// TIA Portal V17 export
// export: Created 2022-01-31T14:44:44.9197147Z, ExportSetting WithDefaults, DisplayName Totally Integrated Automation Portal, DisplayVersion V17, DisplayName TIA Portal Openness, DisplayVersion V17, DisplayName TIA Portal Version Control Interface, DisplayVersion V17, DisplayName STEP 7 Professional, DisplayVersion V17, DisplayName STEP 7 Safety, DisplayVersion V17, DisplayName WinCC Professional, DisplayVersion V17
DATA_BLOCK "FB_Condensador_DB"   // DB8
VERSION : 0.1
// stored: AutoNumber true, DBAccessibleFromOPCUA true, DBAccessibleFromWebserver true, InstanceOfName FB_Condensador, InstanceOfType FB
"FB_Condensador"
   // VAR_OUTPUT
   //    oActual : Int;
   //    oTimer1Min : Int;
   //    oTimer15Sec : Int;
   //    oTimer5Sec : Int;
   // END_VAR
   // VAR
   //    Timer_1Minuto : TON_TIME;
   //    Timer_15sec { S7_SetPoint := 'True'} : TON_TIME;
   //    Timer_5Sec { S7_SetPoint := 'True'} : TON_TIME;
   // END_VAR
BEGIN
END_DATA_BLOCK
